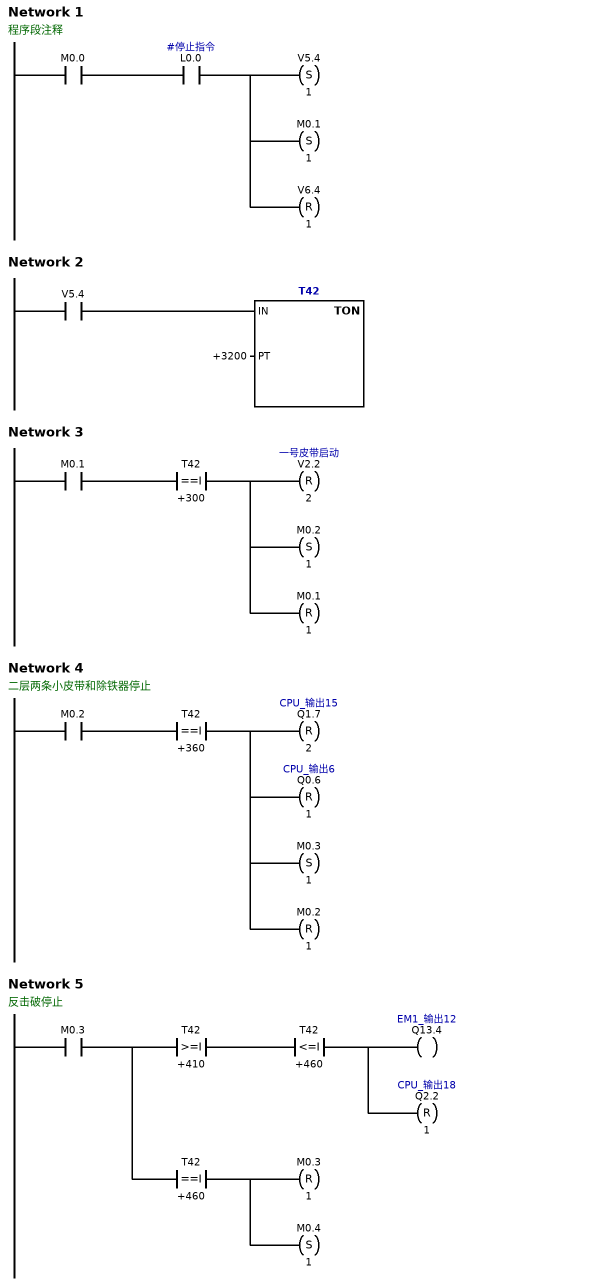
[picture p24: SBR7 networks 1-5]
Network 1
// 程序段注释
LD     M0.0
A      #停止指令:L0.0
S      V5.4, 1
S      M0.1, 1
R      V6.4, 1
Network 2
LD     V5.4
TON    T42, +3200
Network 3
LD     M0.1
AW=    T42, +300
R      一号皮带启动:V2.2, 2
S      M0.2, 1
R      M0.1, 1
Network 4
// 二层两条小皮带和除铁器停止
LD     M0.2
AW=    T42, +360
R      CPU_输出15:Q1.7, 2
R      CPU_输出6:Q0.6, 1
S      M0.3, 1
R      M0.2, 1
Network 5
// 反击破停止
LD     M0.3
LPS
AW>=   T42, +410
AW<=   T42, +460
=      EM1_输出12:Q13.4
R      CPU_输出18:Q2.2, 1
LPP
AW=    T42, +460
R      M0.3, 1
S      M0.4, 1
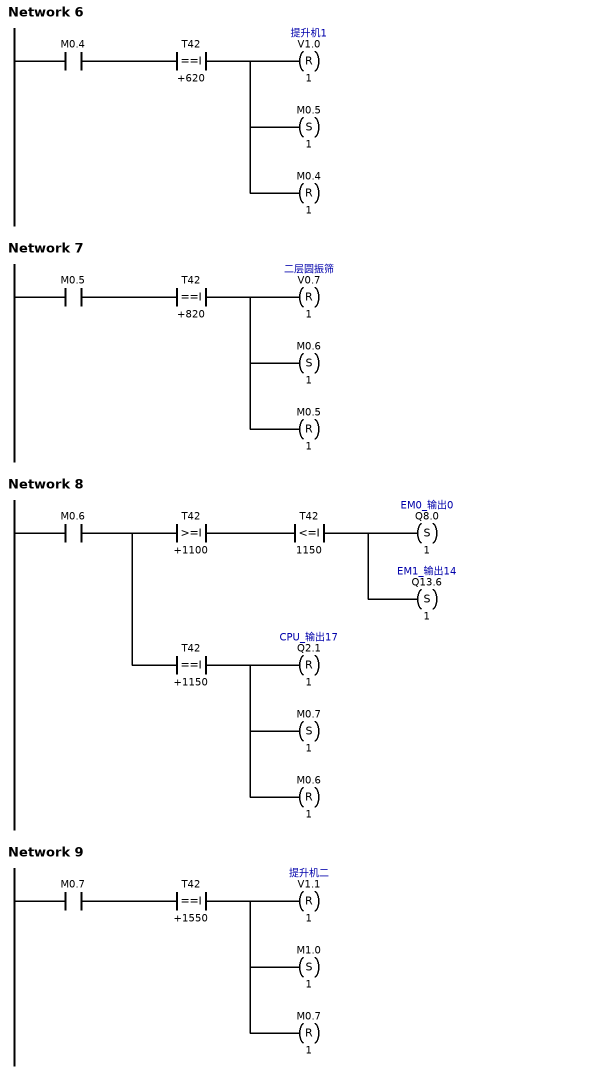
Network 6
LD     M0.4
AW=    T42, +620
R      提升机1:V1.0, 1
S      M0.5, 1
R      M0.4, 1
Network 7
LD     M0.5
AW=    T42, +820
R      二层圆振筛:V0.7, 1
S      M0.6, 1
R      M0.5, 1
Network 8
LD     M0.6
LPS
AW>=   T42, +1100
AW<=   T42, 1150
S      EM0_输出0:Q8.0, 1
S      EM1_输出14:Q13.6, 1
LPP
AW=    T42, +1150
R      CPU_输出17:Q2.1, 1
S      M0.7, 1
R      M0.6, 1
Network 9
LD     M0.7
AW=    T42, +1550
R      提升机二:V1.1, 1
S      M1.0, 1
R      M0.7, 1
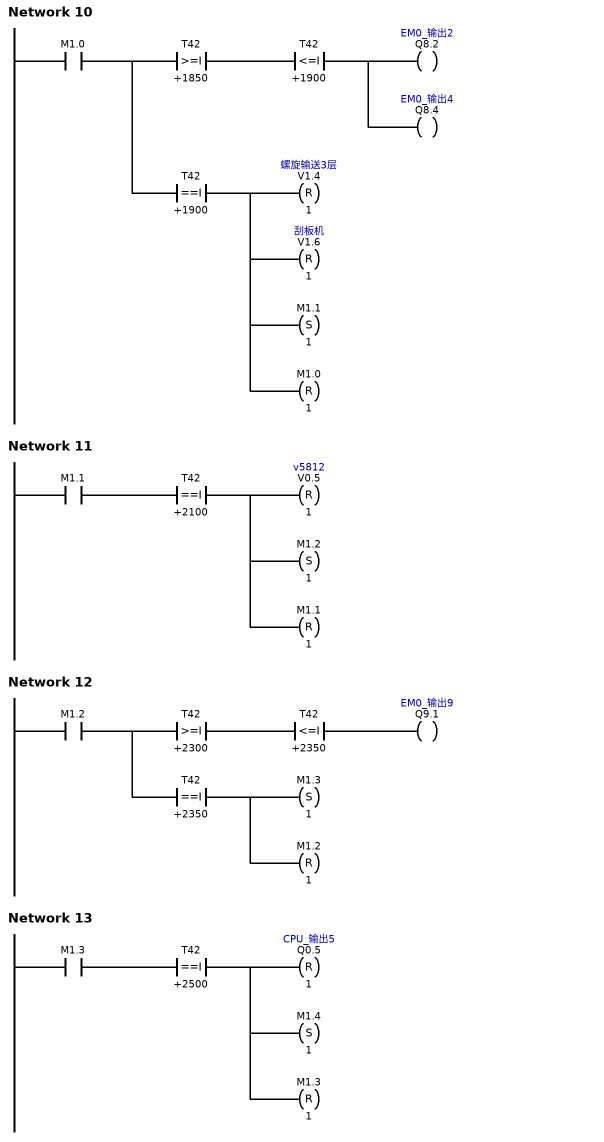
Network 10
LD     M1.0
LPS
AW>=   T42, +1850
AW<=   T42, +1900
=      EM0_输出2:Q8.2
=      EM0_输出4:Q8.4
LPP
AW=    T42, +1900
R      螺旋输送3层:V1.4, 1
R      刮板机:V1.6, 1
S      M1.1, 1
R      M1.0, 1
Network 11
LD     M1.1
AW=    T42, +2100
R      v5812:V0.5, 1
S      M1.2, 1
R      M1.1, 1
Network 12
LD     M1.2
LPS
AW>=   T42, +2300
AW<=   T42, +2350
=      EM0_输出9:Q9.1
LPP
AW=    T42, +2350
S      M1.3, 1
R      M1.2, 1
Network 13
LD     M1.3
AW=    T42, +2500
R      CPU_输出5:Q0.5, 1
S      M1.4, 1
R      M1.3, 1
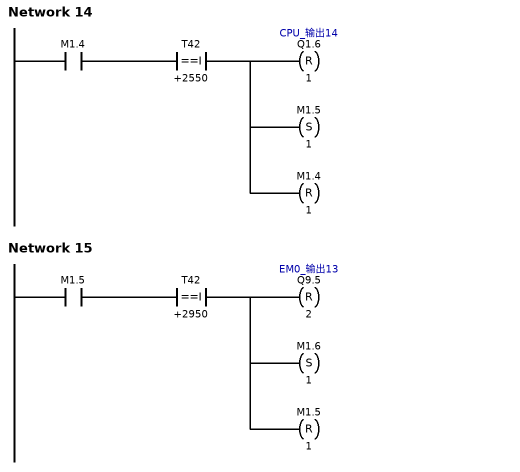
Network 14
LD     M1.4
AW=    T42, +2550
R      CPU_输出14:Q1.6, 1
S      M1.5, 1
R      M1.4, 1
Network 15
LD     M1.5
AW=    T42, +2950
R      EM0_输出13:Q9.5, 2
S      M1.6, 1
R      M1.5, 1
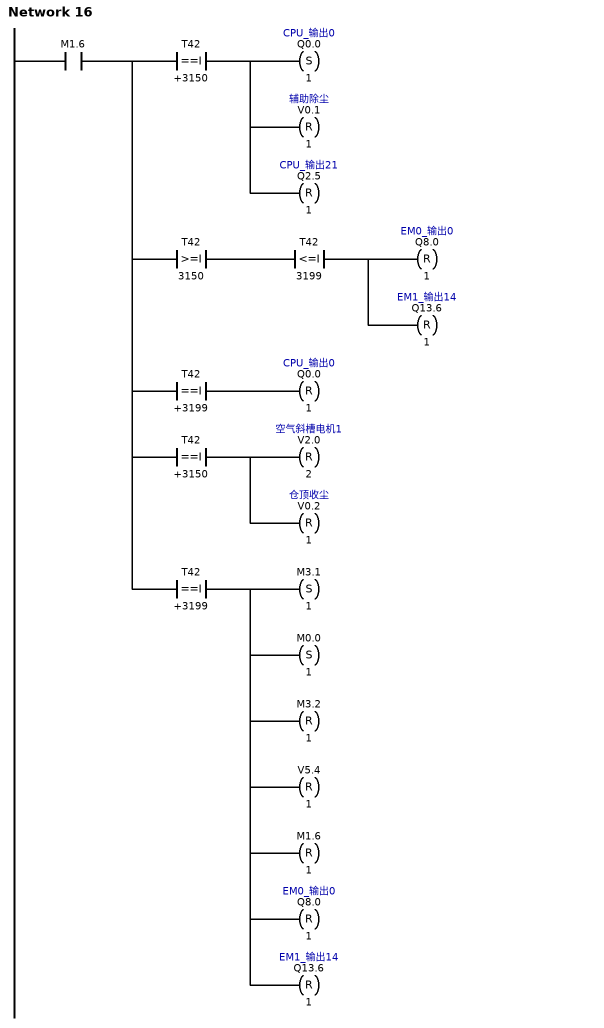
Network 16
LD     M1.6
LPS
AW=    T42, +3150
S      CPU_输出0:Q0.0, 1
R      辅助除尘:V0.1, 1
R      CPU_输出21:Q2.5, 1
LRD
AW>=   T42, 3150
AW<=   T42, 3199
R      EM0_输出0:Q8.0, 1
R      EM1_输出14:Q13.6, 1
LRD
AW=    T42, +3199
R      CPU_输出0:Q0.0, 1
LRD
AW=    T42, +3150
R      空气斜槽电机1:V2.0, 2
R      仓顶收尘:V0.2, 1
LPP
AW=    T42, +3199
S      M3.1, 1
S      M0.0, 1
R      M3.2, 1
R      V5.4, 1
R      M1.6, 1
R      EM0_输出0:Q8.0, 1
R      EM1_输出14:Q13.6, 1
END_SUBROUTINE_BLOCK

SUBROUTINE_BLOCK 急停呦:SBR8
TITLE=子程序注释
VAR_INPUT
急停:BOOL;	// L0.0 
END_VAR
BEGIN
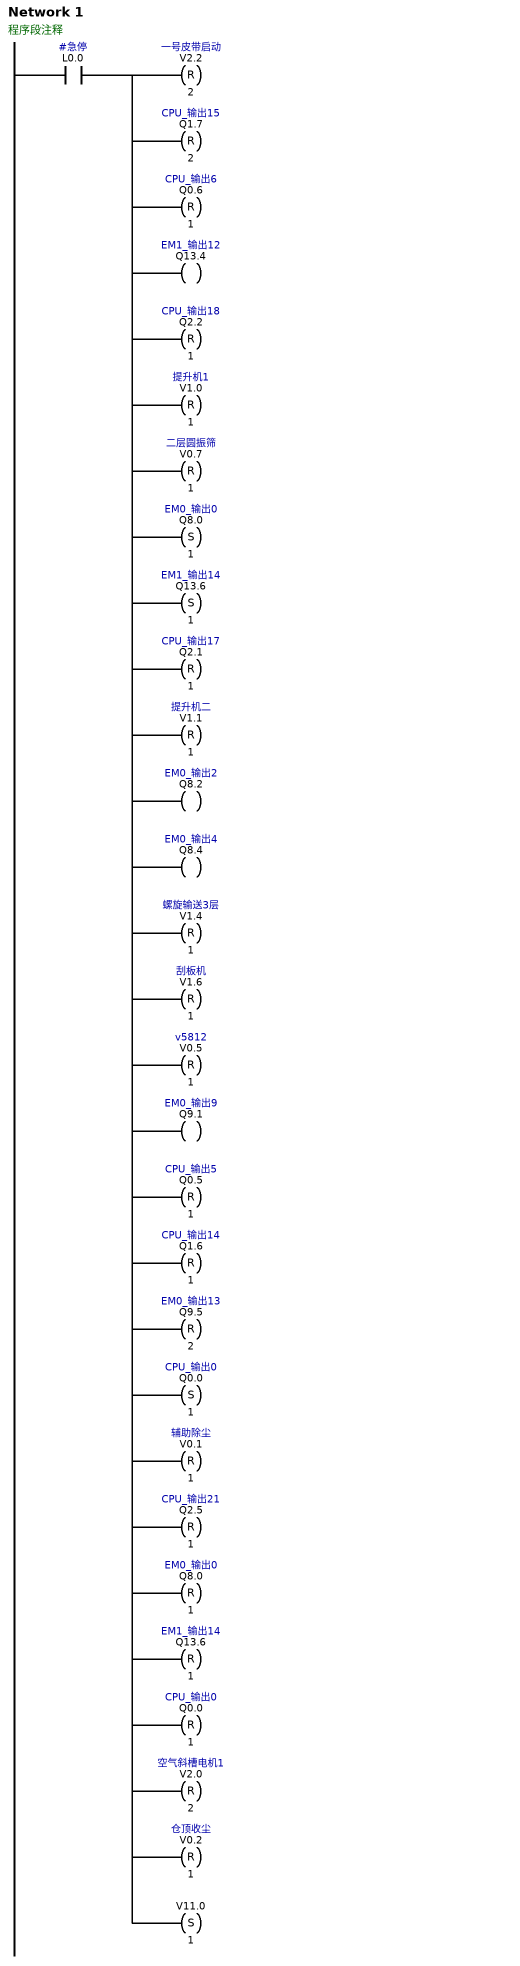
Network 1
// 程序段注释
LD     #急停:L0.0
R      一号皮带启动:V2.2, 2
R      CPU_输出15:Q1.7, 2
R      CPU_输出6:Q0.6, 1
=      EM1_输出12:Q13.4
R      CPU_输出18:Q2.2, 1
R      提升机1:V1.0, 1
R      二层圆振筛:V0.7, 1
S      EM0_输出0:Q8.0, 1
S      EM1_输出14:Q13.6, 1
R      CPU_输出17:Q2.1, 1
R      提升机二:V1.1, 1
=      EM0_输出2:Q8.2
=      EM0_输出4:Q8.4
R      螺旋输送3层:V1.4, 1
R      刮板机:V1.6, 1
R      v5812:V0.5, 1
=      EM0_输出9:Q9.1
R      CPU_输出5:Q0.5, 1
R      CPU_输出14:Q1.6, 1
R      EM0_输出13:Q9.5, 2
S      CPU_输出0:Q0.0, 1
R      辅助除尘:V0.1, 1
R      CPU_输出21:Q2.5, 1
R      EM0_输出0:Q8.0, 1
R      EM1_输出14:Q13.6, 1
R      CPU_输出0:Q0.0, 1
R      空气斜槽电机1:V2.0, 2
R      仓顶收尘:V0.2, 1
S      V11.0, 1
END_SUBROUTINE_BLOCK
